(* Schneider Machine Expert - Basic project zbiornik -- 1.3, file version 2.2.0.0 *)
(* ProjectInformations: Name=Training project, Description=Woda do napełnienia zbiornika ZB1 jest pompowana przez pompę P1, a następnie wylewana przez zawór Z1. Ilość wylewanej wody nie jest stała, jest regulowana ręczne przez Operatora zbiorniku (prawdopodobnie, zgodnie z żądaniami konsumentów).
Aby uniknąć przepełnienia zbiornika i / lub opróżniania rury, zbiornik jest wyposażony w czujniki minimalnego i maksymalnego poziomu wody.
-----
Warunki początkowe: zbiornik wody jest pusty, zawór wyboru wody jest zamknięty.
Urządzenie włącza się, naciskając przycisk START. Pompa dostarcza wodę do zbiornika. Po osiągnięciu poziomu „min-up” otwiera się zawór wylewania wody. Jeżeli pobór wody przekroczy natężenie przepływu, zawór zamknie się ponownie po osiągnięciu poziomu „min-down”. W przeciwnym razie zbiornik będzie nadal napełniany wodą, a gdy poziom osiągnie poziom „max-up”, pompa wyłączy się, a zawór pozostanie otwarty. Pompa włączy się ponowie, gdy osiągnie „max-down” poziom.
Operator może ręcznie zmienić przepustowość zaworu, podczas gdy układ sterowania nie pozwala na przelanie się zbiornika i / lub ewentualne uszkodzenie urządzenia w wyniku nagłej utraty wody w odprowadzanym rurociągu.
Naciśnięcie przycisku STOP powoduje wyłączenie pompy i zamknięcie zaworu. *)
(* UserInformations: LastName=Melnychenko, FirstName=Dmytro, Email=melnyczenko@poczta.pl, Country=Poland *)

HARDWARE
  Cpu 0: TM221M16R/G
  EthernetConfiguration: NetworkName=M221, IpAllocationMode=FixedAddress, IpAddress=0.0.0.0, SubnetMask=0.0.0.0
  SerialLineConfiguration: Baud=Baud19200, Parity=ParityEven, DataBits=DataBits8, StopBits=StopBits1, PhysicalMedium=PhysicalMediumRs485, SlaveId=1, Addressing=SlaveAddressing
  MastTask: UsePeriodScanMode=false, PeriodScan=100
  FastTask: Period=255
  CpuBehavior: StartingMode=StartAsPreviousState, AutoSaveRamOnEeprom=true, WatchdogPeriod=250

SYMBOLS  (address, symbol, comment, settings)
  %M100     M_100  "RUN Relay"
  %M101     M_101  "STOP Relay"
  %M103     M_103  "Czujnik: MIN (Suchobieg)"
  %M104     M_104  "Czujnik: MAX"
  %M105     M_105  "Praca ("1") -- Test ("0")"
  %M106     M_106  "Zawór odpływu ("1" -- otwarty)"
  %M107     M_107  "Silnik pompy ("1" -- praca)"
  %M123     M_123  "Stan czujnika MIN"
  %M124     M_124  "Stan czujnika MAX"
  %S6       SB_TB1S  "Time base of 1 s generated by an internal clock"
  %S13      SB_FIRSTRUN  "Indicates the first controller cycle in RUN mode"
  %MW108    MW_108  "Wydajność zaworu (wylewanie)"
  %MW109    MW_109  "Wydajność pompy (tłoczenie)"
  %MW110    MW_110  "Bieżący poziom wody"
  %MW111    MW_111  "Górny limit czyjnika MAX"
  %MW112    MW_112  "Dolny limit czujnika MAX"
  %MW113    MW_113  "Górny limit czujnika MIN"
  %MW114    MW_114  "Dolny limit czujnika MIN"
  %I0.3     I_0_3  "Suchobieg"
  %I0.4     I_0_4  "Max poziom"
  %I0.5     I_0_5  "PRACA - TEST"
  %I0.6     I_0_6  "STOP"
  %I0.7     I_0_7  "START"
  %Q0.6     Q_0_6  "Sterowanie zaworem odpływu wody"
  %Q0.7     Q_0_7  "Sterowanie pracą pompy"
  %IW0.0    IW_0_0  "Wydajność zaworu"  [Type=Type_0_10V, Scope=Scope_Normal, Minimum=0, Maximum=1000]
  %IW0.1    IW_0_1  "Wydajność pompy"  [Type=Type_0_10V, Scope=Scope_Normal, Minimum=0, Maximum=1000]

POU Kontrola
  (* SectionNumber=1 *)

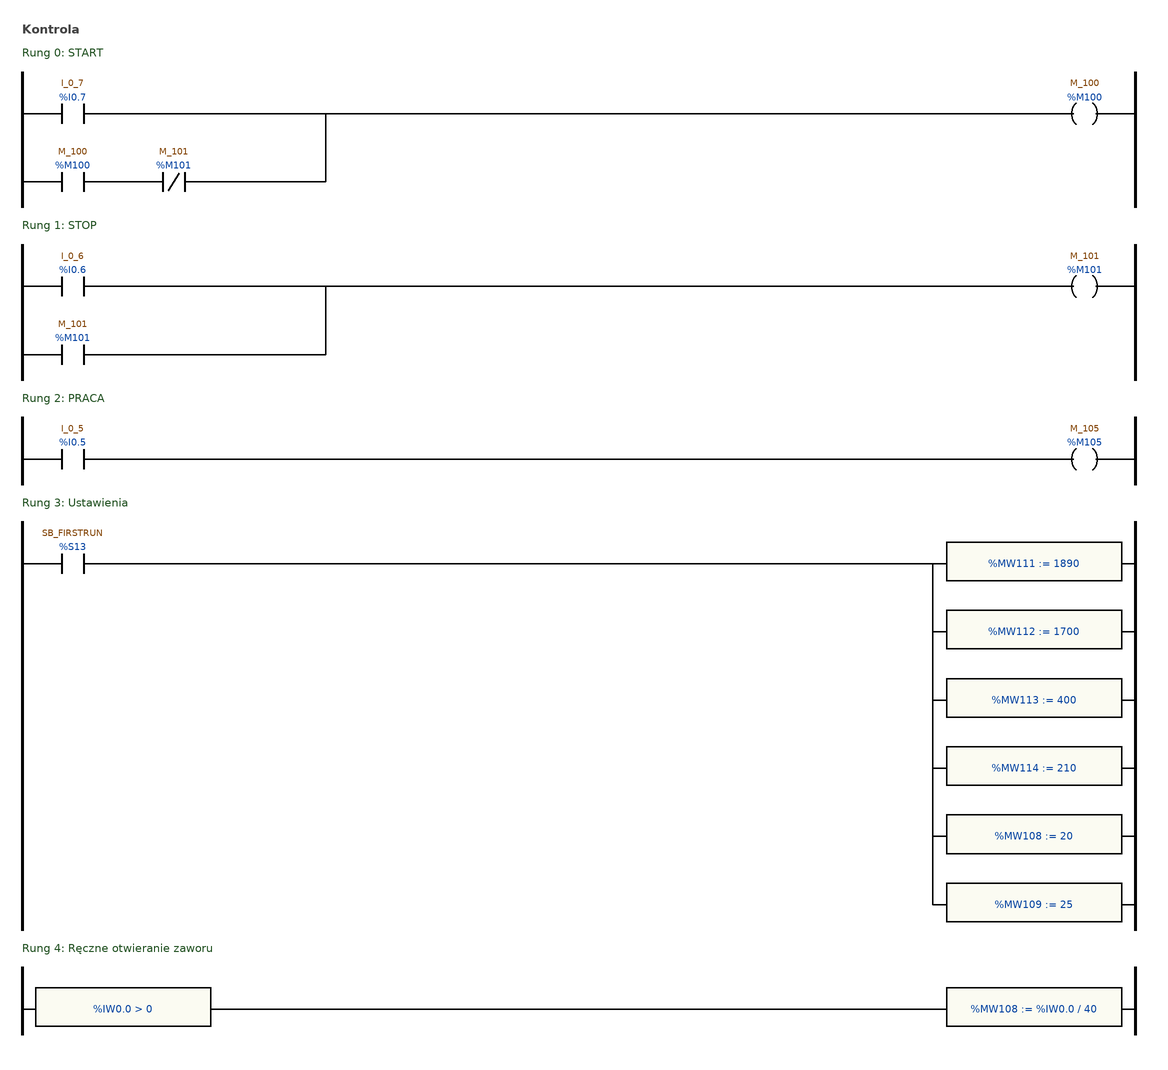

// Rung 0: START
  LD %I0.7                (* I_0_7 *)
  OR( %M100               (* M_100 *)
  ANDN %M101              (* M_101 *)
  )
  ST %M100                (* M_100 *)
  // as ST:
  //   M_100 := I_0_7 OR M_100 AND NOT M_101;

// Rung 1: STOP
  LD %I0.6                (* I_0_6 *)
  OR %M101                (* M_101 *)
  ST %M101                (* M_101 *)
  // as ST:
  //   M_101 := I_0_6 OR M_101;

// Rung 2: PRACA
  LD %I0.5                (* I_0_5 *)
  ST %M105                (* M_105 *)
  // as ST:
  //   M_105 := I_0_5;

// Rung 3: Ustawienia
  LD %S13                 (* SB_FIRSTRUN *)
  [ %MW111 := 1890 ]      (* MW_111 *)
  [ %MW112 := 1700 ]      (* MW_112 *)
  [ %MW113 := 400 ]       (* MW_113 *)
  [ %MW114 := 210 ]       (* MW_114 *)
  [ %MW108 := 20 ]        (* MW_108 *)
  [ %MW109 := 25 ]        (* MW_109 *)
  // as ST:
  //   IF SB_FIRSTRUN THEN MW_111 := 1890; END_IF;
  //   IF SB_FIRSTRUN THEN MW_112 := 1700; END_IF;
  //   IF SB_FIRSTRUN THEN MW_113 := 400; END_IF;
  //   IF SB_FIRSTRUN THEN MW_114 := 210; END_IF;
  //   IF SB_FIRSTRUN THEN MW_108 := 20; END_IF;
  //   IF SB_FIRSTRUN THEN MW_109 := 25; END_IF;

// Rung 4: Ręczne otwieranie zaworu
  LD [ %IW0.0 > 0 ]       (* IW_0_0 *)
  [ %MW108 := %IW0.0 / 40 ](* MW_108, IW_0_0 *)
  // as ST:
  //   IF IW_0_0 > 0 THEN MW_108 := IW_0_0 / 40; END_IF;

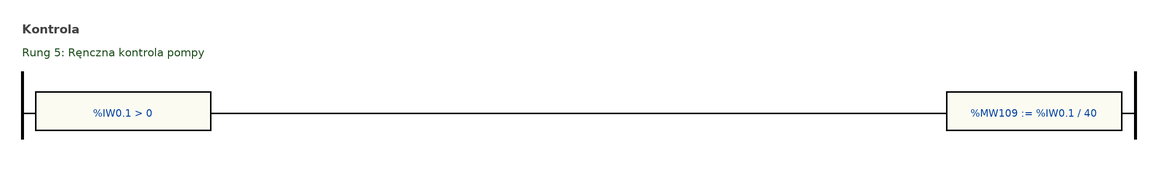

// Rung 5: Ręnczna kontrola pompy
  LD [ %IW0.1 > 0 ]       (* IW_0_1 *)
  [ %MW109 := %IW0.1 / 40 ](* MW_109, IW_0_1 *)
  // as ST:
  //   IF IW_0_1 > 0 THEN MW_109 := IW_0_1 / 40; END_IF;

POU Sterowanie pompą i zaworem
  (* SectionNumber=2 *)

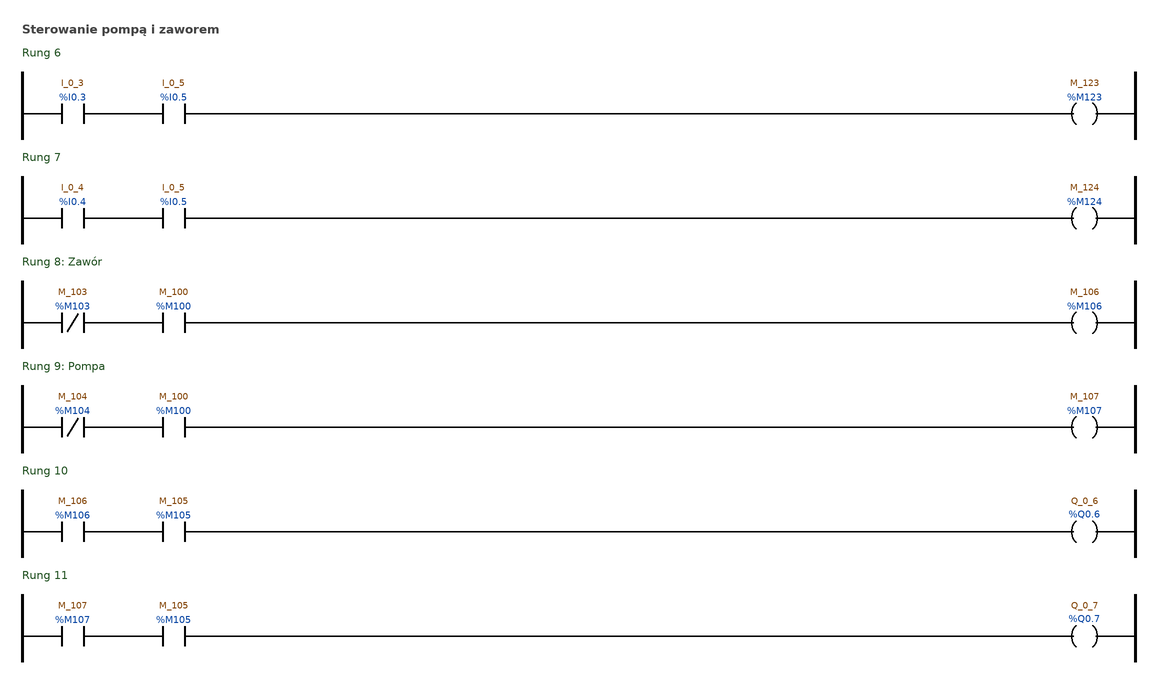

// Rung 6
  LD %I0.3                (* I_0_3 *)
  AND %I0.5               (* I_0_5 *)
  ST %M123                (* M_123 *)
  // as ST:
  //   M_123 := I_0_3 AND I_0_5;

// Rung 7
  LD %I0.4                (* I_0_4 *)
  AND %I0.5               (* I_0_5 *)
  ST %M124                (* M_124 *)
  // as ST:
  //   M_124 := I_0_4 AND I_0_5;

// Rung 8: Zawór
  LDN %M103               (* M_103 *)
  AND %M100               (* M_100 *)
  ST %M106                (* M_106 *)
  // as ST:
  //   M_106 := NOT M_103 AND M_100;

// Rung 9: Pompa
  LDN %M104               (* M_104 *)
  AND %M100               (* M_100 *)
  ST %M107                (* M_107 *)
  // as ST:
  //   M_107 := NOT M_104 AND M_100;

// Rung 10
  LD %M106                (* M_106 *)
  AND %M105               (* M_105 *)
  ST %Q0.6                (* Q_0_6 *)
  // as ST:
  //   Q_0_6 := M_106 AND M_105;

// Rung 11
  LD %M107                (* M_107 *)
  AND %M105               (* M_105 *)
  ST %Q0.7                (* Q_0_7 *)
  // as ST:
  //   Q_0_7 := M_107 AND M_105;

POU Emulator tłoczenia i wylewania
  (* SectionNumber=3 *)

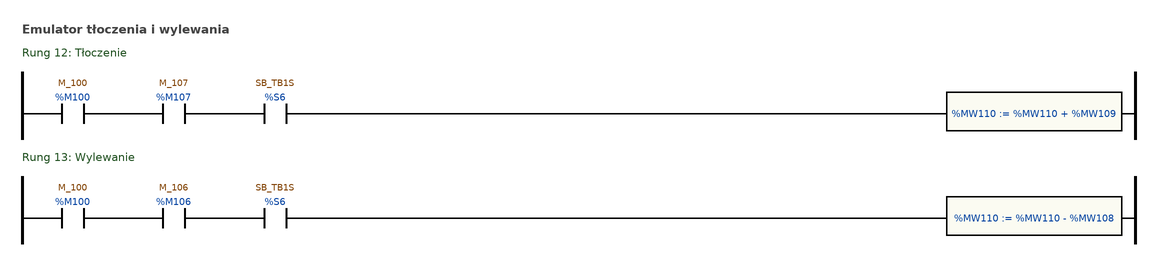

// Rung 12: Tłoczenie
  LD %M100                (* M_100 *)
  AND %M107               (* M_107 *)
  AND %S6                 (* SB_TB1S *)
  [ %MW110 := %MW110 + %MW109 ](* MW_110, MW_110, MW_109 *)
  // as ST:
  //   IF M_100 AND M_107 AND SB_TB1S THEN MW_110 := MW_110 + MW_109; END_IF;

// Rung 13: Wylewanie
  LD %M100                (* M_100 *)
  AND %M106               (* M_106 *)
  AND %S6                 (* SB_TB1S *)
  [ %MW110 := %MW110 - %MW108 ](* MW_110, MW_110, MW_108 *)
  // as ST:
  //   IF M_100 AND M_106 AND SB_TB1S THEN MW_110 := MW_110 - MW_108; END_IF;

POU Emulator Histerezy Pływaków
  (* SectionNumber=4 *)

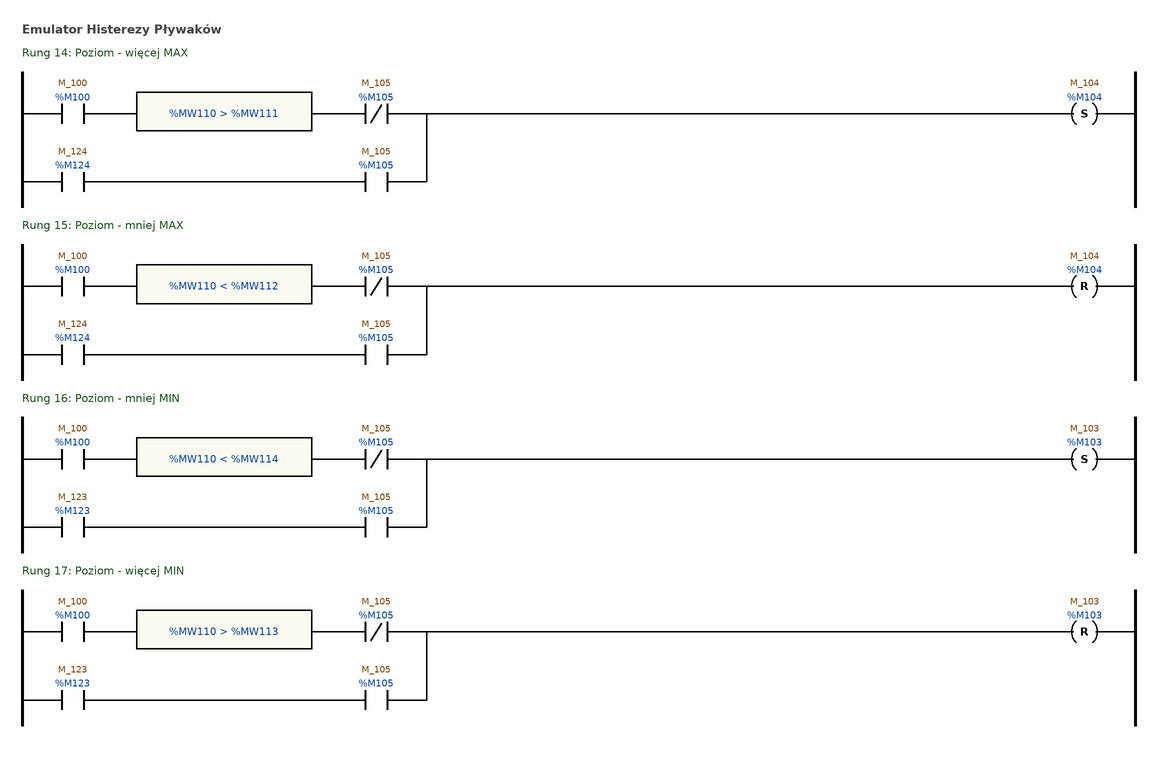

// Rung 14: Poziom - więcej MAX
  LD %M100                (* M_100 *)
  AND [ %MW110 > %MW111 ] (* MW_110, MW_111 *)
  ANDN %M105              (* M_105 *)
  OR( %M124               (* M_124 *)
  AND %M105               (* M_105 *)
  )
  S %M104                 (* M_104 *)
  // as ST:
  //   IF M_100 AND MW_110 > MW_111 AND NOT M_105 OR M_124 AND M_105 THEN M_104 := TRUE; END_IF;

// Rung 15: Poziom - mniej MAX
  LD %M100                (* M_100 *)
  AND [ %MW110 < %MW112 ] (* MW_110, MW_112 *)
  ANDN %M105              (* M_105 *)
  OR( %M124               (* M_124 *)
  AND %M105               (* M_105 *)
  )
  R %M104                 (* M_104 *)
  // as ST:
  //   IF M_100 AND MW_110 < MW_112 AND NOT M_105 OR M_124 AND M_105 THEN M_104 := FALSE; END_IF;

// Rung 16: Poziom - mniej MIN
  LD %M100                (* M_100 *)
  AND [ %MW110 < %MW114 ] (* MW_110, MW_114 *)
  ANDN %M105              (* M_105 *)
  OR( %M123               (* M_123 *)
  AND %M105               (* M_105 *)
  )
  S %M103                 (* M_103 *)
  // as ST:
  //   IF M_100 AND MW_110 < MW_114 AND NOT M_105 OR M_123 AND M_105 THEN M_103 := TRUE; END_IF;

// Rung 17: Poziom - więcej MIN
  LD %M100                (* M_100 *)
  AND [ %MW110 > %MW113 ] (* MW_110, MW_113 *)
  ANDN %M105              (* M_105 *)
  OR( %M123               (* M_123 *)
  AND %M105               (* M_105 *)
  )
  R %M103                 (* M_103 *)
  // as ST:
  //   IF M_100 AND MW_110 > MW_113 AND NOT M_105 OR M_123 AND M_105 THEN M_103 := FALSE; END_IF;
